// TwinCAT 3 PLC project T1SchmittTrigger_Plc
// Title: T1SchmittTrigger_Plc
// Company: Tc3 Project
// ProjectVersion: 1.0.0.0
// ProgramVersion: 3.1.4026.22
// libraries:
//   Tc2_Standard, * (Beckhoff Automation GmbH)
//   Tc2_System, * (Beckhoff Automation GmbH)
// project tree:
//   / PlcTask.TcTTO
//   POUs/ FB_SchmittTrigger.TcPOU, MAIN.TcPOU
// real-time tasks:
//   TASK PlcTask: cycle T#10ms, priority 20, ADS port 350

CONFIGURATION T1SchmittTrigger_Plc
    RESOURCE PLC ON TwinCAT3
        TASK PlcTask(INTERVAL := T#10ms, PRIORITY := 20);
        PROGRAM MAIN WITH PlcTask : MAIN;
    END_RESOURCE
END_CONFIGURATION

// ---- POUs/MAIN.TcPOU
PROGRAM MAIN
VAR
END_VAR

END_PROGRAM

// ---- POUs/FB_SchmittTrigger.TcPOU
FUNCTION_BLOCK FB_SchmittTrigger
VAR_INPUT
    fInput : REAL;
    fLowThreshold : REAL := 0.3;
    fHighThreshold : REAL := 0.7;
END_VAR
VAR_OUTPUT
    bState : BOOL;
END_VAR

METHOD Step : BOOL
;
END_METHOD

END_FUNCTION_BLOCK
